{attribute 'qualified_only'}
{attribute 'strict'}
(*
TYPE ePowerStatus :
(
	Off := 	0,
	On	:=	1,
	Fault	:=	2
);
*)

(* stored: Version 1.1.0.1, ProductVersion 3.1.4024.12
   DUT ePowerStatus: Id {fb9437b8-d02a-4fea-b938-d9638caaf087} *)
